LIN {X 0,Y 85.092,Z 662.145,A -85,B 0,C 180,E1 -19260,E2 -19260} C_VEL
LIN {X 0,Y 82.848,Z 665.659,A -85,B 0,C 180,E1 -19250.232,E2 -19250.232} C_VEL
LIN {X 0,Y 84.77,Z 669.976,A -85,B 0,C 180,E1 -19235.51,E2 -19235.51} C_VEL
LIN {X 0,Y 86.766,Z 671.167,A -85,B 0,C 180,E1 -19230.922,E2 -19230.922} C_VEL
LIN {X 0,Y 92.025,Z 672.605,A -85,B 0,C 180,E1 -19223.904,E2 -19223.904} C_VEL
LIN {X 0,Y 91.235,Z 673.792,A -85,B 0,C 180,E1 -19222.952,E2 -19222.952} C_VEL
LIN {X 0,Y 83.813,Z 680.743,A -85,B 0,C 180,E1 -19217.869,E2 -19217.869} C_VEL
LIN {X 0,Y 77.915,Z 685.734,A -85,B 0,C 180,E1 -19212.572,E2 -19212.572} C_VEL
LIN {X 0,Y 72.15,Z 690.144,A -85,B 0,C 180,E1 -19205.764,E2 -19205.764} C_VEL
LIN {X 0,Y 68.908,Z 692.468,A -85,B 0,C 180,E1 -19200.661,E2 -19200.661} C_VEL
LIN {X 0,Y 66.35,Z 694.368,A -85,B 0,C 180,E1 -19195.068,E2 -19195.068} C_VEL
LIN {X 0,Y 64.456,Z 695.815,A -85,B 0,C 180,E1 -19189.093,E2 -19189.093} C_VEL
LIN {X 0,Y 63.195,Z 696.835,A -85,B 0,C 180,E1 -19182.851,E2 -19182.851} C_VEL
LIN {X 0,Y 62.592,Z 697.466,A -85,B 0,C 180,E1 -19176.447,E2 -19176.447} C_VEL
LIN {X 0,Y 62.642,Z 697.705,A -85,B 0,C 180,E1 -19170,E2 -19170} C_VEL
LIN {X 0,Y 62.755,Z 697.489,A -85,B 0,C 180,E1 -19163.57,E2 -19163.57} C_VEL
LIN {X 0,Y 64.913,Z 695.872,A -85,B 0,C 180,E1 -19151.046,E2 -19151.046} C_VEL
LIN {X 0,Y 67.088,Z 694.459,A -85,B 0,C 180,E1 -19145.226,E2 -19145.226} C_VEL
LIN {X 0,Y 71.596,Z 691.514,A -85,B 0,C 180,E1 -19137.324,E2 -19137.324} C_VEL
LIN {X 0,Y 77.419,Z 687.523,A -85,B 0,C 180,E1 -19130.546,E2 -19130.546} C_VEL
LIN {X 0,Y 84.572,Z 682.371,A -85,B 0,C 180,E1 -19125.06,E2 -19125.06} C_VEL
LIN {X 0,Y 87.182,Z 680.379,A -85,B 0,C 180,E1 -19123.488,E2 -19123.488} C_VEL
LIN {X 0,Y 82.264,Z 678.447,A -85,B 0,C 180,E1 -19116.729,E2 -19116.729} C_VEL
LIN {X 0,Y 79.03,Z 677.694,A -85,B 0,C 180,E1 -19112.247,E2 -19112.247} C_VEL
LIN {X 0,Y 76.795,Z 676.602,A -85,B 0,C 180,E1 -19107.231,E2 -19107.231} C_VEL
LIN {X 0,Y 75.533,Z 675.043,A -85,B 0,C 180,E1 -19101.494,E2 -19101.494} C_VEL
LIN {X 0,Y 74.478,Z 672.702,A -85,B 0,C 180,E1 -19090.878,E2 -19090.878} C_VEL
LIN {X 0,Y 76.565,Z 669.743,A -85,B 0,C 180,E1 -19080,E2 -19080} C_VEL
LIN {X 0,Y 83.879,Z 665.425,A -85,B 0,C 180,E1 -19065.442,E2 -19065.442} C_VEL
LIN {X 0,Y 96.513,Z 659.738,A -85,B 0,C 180,E1 -19054.092,E2 -19054.092} C_VEL
LIN {X 0,Y 99.35,Z 658.243,A -85,B 0,C 180,E1 -19052.625,E2 -19052.625} C_VEL
LIN {X 0,Y 105.136,Z 655.722,A -85,B 0,C 180,E1 -19049.405,E2 -19049.405} C_VEL
LIN {X 0,Y 105.017,Z 656.515,A -85,B 0,C 180,E1 -19048.696,E2 -19048.696} C_VEL
LIN {X 0,Y 98.158,Z 664.839,A -85,B 0,C 180,E1 -19045.426,E2 -19045.426} C_VEL
LIN {X 0,Y 90.491,Z 672.846,A -85,B 0,C 180,E1 -19040.955,E2 -19040.955} C_VEL
LIN {X 0,Y 83.376,Z 679.286,A -85,B 0,C 180,E1 -19035.766,E2 -19035.766} C_VEL
LIN {X 0,Y 76.898,Z 684.398,A -85,B 0,C 180,E1 -19029.774,E2 -19029.774} C_VEL
LIN {X 0,Y 71.412,Z 688.419,A -85,B 0,C 180,E1 -19022.496,E2 -19022.496} C_VEL
LIN {X 0,Y 68.389,Z 690.108,A -85,B 0,C 180,E1 -19018.544,E2 -19018.544} C_VEL
LIN {X 0,Y 62.458,Z 692.322,A -85,B 0,C 180,E1 -19011.839,E2 -19011.839} C_VEL
LIN {X 0,Y 58.208,Z 693.565,A -85,B 0,C 180,E1 -19005.545,E2 -19005.545} C_VEL
LIN {X 0,Y 56.215,Z 694.173,A -85,B 0,C 180,E1 -18999.984,E2 -18999.984} C_VEL
LIN {X 0,Y 55.916,Z 694.293,A -85,B 0,C 180,E1 -18997.996,E2 -18997.996} C_VEL
LIN {X 0,Y 55.609,Z 694.556,A -85,B 0,C 180,E1 -18990,E2 -18990} C_VEL
LIN {X 0,Y 56.865,Z 693.723,A -85,B 0,C 180,E1 -18975.689,E2 -18975.689} C_VEL
LIN {X 0,Y 58.571,Z 692.733,A -85,B 0,C 180,E1 -18968.901,E2 -18968.901} C_VEL
LIN {X 0,Y 60.958,Z 691.321,A -85,B 0,C 180,E1 -18962.537,E2 -18962.537} C_VEL
LIN {X 0,Y 65.7,Z 688.393,A -85,B 0,C 180,E1 -18953.961,E2 -18953.961} C_VEL
LIN {X 0,Y 71.617,Z 684.415,A -85,B 0,C 180,E1 -18946.612,E2 -18946.612} C_VEL
LIN {X 0,Y 78.615,Z 679.262,A -85,B 0,C 180,E1 -18940.546,E2 -18940.546} C_VEL
LIN {X 0,Y 86.232,Z 672.778,A -85,B 0,C 180,E1 -18935.412,E2 -18935.412} C_VEL
LIN {X 0,Y 94.349,Z 664.71,A -85,B 0,C 180,E1 -18931.059,E2 -18931.059} C_VEL
LIN {X 0,Y 101.472,Z 656.423,A -85,B 0,C 180,E1 -18927.984,E2 -18927.984} C_VEL
LIN {X 0,Y 105.069,Z 651.685,A -85,B 0,C 180,E1 -18926.643,E2 -18926.643} C_VEL
LIN {X 0,Y 105.974,Z 649.829,A -85,B 0,C 180,E1 -18925.697,E2 -18925.697} C_VEL
LIN {X 0,Y 97.243,Z 655.594,A -85,B 0,C 180,E1 -18921.184,E2 -18921.184} C_VEL
LIN {X 0,Y 92.45,Z 658.477,A -85,B 0,C 180,E1 -18917.703,E2 -18917.703} C_VEL
LIN {X 0,Y 88.64,Z 660.634,A -85,B 0,C 180,E1 -18913.761,E2 -18913.761} C_VEL
LIN {X 0,Y 85.467,Z 662.497,A -85,B 0,C 180,E1 -18909.466,E2 -18909.466} C_VEL
LIN {X 0,Y 80.521,Z 666.215,A -85,B 0,C 180,E1 -18902.501,E2 -18902.501} C_VEL
LIN {X 0,Y 77.739,Z 669.133,A -85,B 0,C 180,E1 -18893.966,E2 -18893.966} C_VEL
LIN {X 0,Y 80.998,Z 675.167,A -85,B 0,C 180,E1 -18870.191,E2 -18870.191} C_VEL
LIN {X 0,Y 83.783,Z 675.989,A -85,B 0,C 180,E1 -18865.868,E2 -18865.868} C_VEL
LIN {X 0,Y 82.502,Z 677.724,A -85,B 0,C 180,E1 -18864.025,E2 -18864.025} C_VEL
LIN {X 0,Y 75.151,Z 683.798,A -85,B 0,C 180,E1 -18858.431,E2 -18858.431} C_VEL
LIN {X 0,Y 68.463,Z 688.599,A -85,B 0,C 180,E1 -18851.856,E2 -18851.856} C_VEL
LIN {X 0,Y 62.89,Z 692.278,A -85,B 0,C 180,E1 -18843.97,E2 -18843.97} C_VEL
LIN {X 0,Y 59.952,Z 694.177,A -85,B 0,C 180,E1 -18837.964,E2 -18837.964} C_VEL
LIN {X 0,Y 57.765,Z 695.625,A -85,B 0,C 180,E1 -18831.408,E2 -18831.408} C_VEL
LIN {X 0,Y 56.28,Z 696.646,A -85,B 0,C 180,E1 -18824.463,E2 -18824.463} C_VEL
LIN {X 0,Y 55.542,Z 697.277,A -85,B 0,C 180,E1 -18817.269,E2 -18817.269} C_VEL
LIN {X 0,Y 55.532,Z 697.516,A -85,B 0,C 180,E1 -18810,E2 -18810} C_VEL
LIN {X 0,Y 55.692,Z 697.3,A -85,B 0,C 180,E1 -18802.75,E2 -18802.75} C_VEL
LIN {X 0,Y 58.239,Z 695.683,A -85,B 0,C 180,E1 -18788.775,E2 -18788.775} C_VEL
LIN {X 0,Y 60.713,Z 694.271,A -85,B 0,C 180,E1 -18782.417,E2 -18782.417} C_VEL
LIN {X 0,Y 65.745,Z 691.327,A -85,B 0,C 180,E1 -18773.989,E2 -18773.989} C_VEL
LIN {X 0,Y 72.078,Z 687.336,A -85,B 0,C 180,E1 -18766.958,E2 -18766.958} C_VEL
LIN {X 0,Y 78.39,Z 683.096,A -85,B 0,C 180,E1 -18762.238,E2 -18762.238} C_VEL
LIN {X 0,Y 78.058,Z 682.451,A -85,B 0,C 180,E1 -18760.697,E2 -18760.697} C_VEL
LIN {X 0,Y 71.292,Z 680.424,A -85,B 0,C 180,E1 -18749.531,E2 -18749.531} C_VEL
LIN {X 0,Y 72.504,Z 672.841,A -85,B 0,C 180,E1 -18714.437,E2 -18714.437} C_VEL
LIN {X 0,Y 78.276,Z 670.097,A -85,B 0,C 180,E1 -18704.374,E2 -18704.374} C_VEL
LIN {X 0,Y 94.026,Z 663.899,A -85,B 0,C 180,E1 -18690.988,E2 -18690.988} C_VEL
LIN {X 0,Y 95.328,Z 663.283,A -85,B 0,C 180,E1 -18690.369,E2 -18690.369} C_VEL
LIN {X 0,Y 94.903,Z 664.393,A -85,B 0,C 180,E1 -18689.273,E2 -18689.273} C_VEL
LIN {X 0,Y 87.657,Z 671.706,A -85,B 0,C 180,E1 -18685.458,E2 -18685.458} C_VEL
LIN {X 0,Y 81.075,Z 677.49,A -85,B 0,C 180,E1 -18681.276,E2 -18681.276} C_VEL
LIN {X 0,Y 73.843,Z 683,A -85,B 0,C 180,E1 -18675.547,E2 -18675.547} C_VEL
LIN {X 0,Y 67.513,Z 687.308,A -85,B 0,C 180,E1 -18668.652,E2 -18668.652} C_VEL
LIN {X 0,Y 63.94,Z 689.573,A -85,B 0,C 180,E1 -18663.338,E2 -18663.338} C_VEL
LIN {X 0,Y 60.953,Z 691.413,A -85,B 0,C 180,E1 -18657.465,E2 -18657.465} C_VEL
LIN {X 0,Y 58.569,Z 692.792,A -85,B 0,C 180,E1 -18651.099,E2 -18651.099} C_VEL
LIN {X 0,Y 55.916,Z 694.293,A -85,B 0,C 180,E1 -18637.996,E2 -18637.996} C_VEL
LIN {X 0,Y 55.317,Z 694.556,A -85,B 0,C 180,E1 -18633.998,E2 -18633.998} C_VEL
LIN {X 0,Y 53.901,Z 694.702,A -85,B 0,C 180,E1 -18627.956,E2 -18627.956} C_VEL
LIN {X 0,Y 51.663,Z 694.275,A -85,B 0,C 180,E1 -18617.386,E2 -18617.386} C_VEL
LIN {X 0,Y 51.576,Z 693.301,A -85,B 0,C 180,E1 -18608.562,E2 -18608.562} C_VEL
LIN {X 0,Y 52.568,Z 692.593,A -85,B 0,C 180,E1 -18604.386,E2 -18604.386} C_VEL
LIN {X 0,Y 58.152,Z 689.651,A -85,B 0,C 180,E1 -18592.823,E2 -18592.823} C_VEL
LIN {X 0,Y 64.344,Z 686.033,A -85,B 0,C 180,E1 -18584.768,E2 -18584.768} C_VEL
LIN {X 0,Y 71.589,Z 681.293,A -85,B 0,C 180,E1 -18578.245,E2 -18578.245} C_VEL
LIN {X 0,Y 79.553,Z 675.292,A -85,B 0,C 180,E1 -18572.937,E2 -18572.937} C_VEL
LIN {X 0,Y 87.984,Z 667.809,A -85,B 0,C 180,E1 -18568.518,E2 -18568.518} C_VEL
LIN {X 0,Y 94.958,Z 660.558,A -85,B 0,C 180,E1 -18565.594,E2 -18565.594} C_VEL
LIN {X 0,Y 95.736,Z 659.289,A -85,B 0,C 180,E1 -18564.747,E2 -18564.747} C_VEL
LIN {X 0,Y 90.805,Z 661.951,A -85,B 0,C 180,E1 -18561.757,E2 -18561.757} C_VEL
LIN {X 0,Y 87.102,Z 663.828,A -85,B 0,C 180,E1 -18558.83,E2 -18558.83} C_VEL
LIN {X 0,Y 80.808,Z 666.963,A -85,B 0,C 180,E1 -18551.657,E2 -18551.657} C_VEL
LIN {X 0,Y 75.932,Z 670.038,A -85,B 0,C 180,E1 -18545.311,E2 -18545.311} C_VEL
LIN {X 0,Y 73.444,Z 671.868,A -85,B 0,C 180,E1 -18540,E2 -18540} C_VEL
LIN {X 0,Y 72.428,Z 677.195,A -85,B 0,C 180,E1 -18517.162,E2 -18517.162} C_VEL
LIN {X 0,Y 74.052,Z 678.364,A -85,B 0,C 180,E1 -18511.672,E2 -18511.672} C_VEL
LIN {X 0,Y 75.813,Z 679.737,A -85,B 0,C 180,E1 -18506.545,E2 -18506.545} C_VEL
LIN {X 0,Y 68.118,Z 685.355,A -85,B 0,C 180,E1 -18500.697,E2 -18500.697} C_VEL
LIN {X 0,Y 61.161,Z 689.764,A -85,B 0,C 180,E1 -18493.588,E2 -18493.588} C_VEL
LIN {X 0,Y 57.129,Z 692.088,A -85,B 0,C 180,E1 -18487.959,E2 -18487.959} C_VEL
LIN {X 0,Y 53.746,Z 693.986,A -85,B 0,C 180,E1 -18481.537,E2 -18481.537} C_VEL
LIN {X 0,Y 51.176,Z 695.434,A -85,B 0,C 180,E1 -18474.33,E2 -18474.33} C_VEL
LIN {X 0,Y 49.403,Z 696.455,A -85,B 0,C 180,E1 -18466.53,E2 -18466.53} C_VEL
LIN {X 0,Y 48.496,Z 697.087,A -85,B 0,C 180,E1 -18458.333,E2 -18458.333} C_VEL
LIN {X 0,Y 48.443,Z 697.327,A -85,B 0,C 180,E1 -18450,E2 -18450} C_VEL
LIN {X 0,Y 48.649,Z 697.111,A -85,B 0,C 180,E1 -18441.694,E2 -18441.694} C_VEL
LIN {X 0,Y 51.688,Z 695.495,A -85,B 0,C 180,E1 -18425.926,E2 -18425.926} C_VEL
LIN {X 0,Y 54.508,Z 694.083,A -85,B 0,C 180,E1 -18418.953,E2 -18418.953} C_VEL
LIN {X 0,Y 60.142,Z 691.139,A -85,B 0,C 180,E1 -18410.006,E2 -18410.006} C_VEL
LIN {X 0,Y 68.937,Z 685.995,A -85,B 0,C 180,E1 -18401.363,E2 -18401.363} C_VEL
LIN {X 0,Y 69.573,Z 684.914,A -85,B 0,C 180,E1 -18399.083,E2 -18399.083} C_VEL
LIN {X 0,Y 64.877,Z 683.489,A -85,B 0,C 180,E1 -18389.931,E2 -18389.931} C_VEL
LIN {X 0,Y 66.397,Z 676.925,A -85,B 0,C 180,E1 -18353.924,E2 -18353.924} C_VEL
LIN {X 0,Y 74.494,Z 673.684,A -85,B 0,C 180,E1 -18340.636,E2 -18340.636} C_VEL
LIN {X 0,Y 86.317,Z 669.604,A -85,B 0,C 180,E1 -18330.756,E2 -18330.756} C_VEL
LIN {X 0,Y 78.2,Z 676.613,A -85,B 0,C 180,E1 -18326.234,E2 -18326.234} C_VEL
LIN {X 0,Y 71.57,Z 681.48,A -85,B 0,C 180,E1 -18321.774,E2 -18321.774} C_VEL
LIN {X 0,Y 64.309,Z 686.182,A -85,B 0,C 180,E1 -18315.264,E2 -18315.264} C_VEL
LIN {X 0,Y 58.139,Z 689.761,A -85,B 0,C 180,E1 -18307.187,E2 -18307.187} C_VEL
LIN {X 0,Y 54.735,Z 691.601,A -85,B 0,C 180,E1 -18300.904,E2 -18300.904} C_VEL
LIN {X 0,Y 51.998,Z 692.98,A -85,B 0,C 180,E1 -18293.921,E2 -18293.921} C_VEL
LIN {X 0,Y 48.876,Z 694.508,A -85,B 0,C 180,E1 -18278.791,E2 -18278.791} C_VEL
LIN {X 0,Y 48.509,Z 694.745,A -85,B 0,C 180,E1 -18270,E2 -18270} C_VEL
LIN {X 0,Y 48.83,Z 694.52,A -85,B 0,C 180,E1 -18261.725,E2 -18261.725} C_VEL
LIN {X 0,Y 50.014,Z 693.912,A -85,B 0,C 180,E1 -18253.677,E2 -18253.677} C_VEL
LIN {X 0,Y 52.568,Z 692.593,A -85,B 0,C 180,E1 -18244.386,E2 -18244.386} C_VEL
LIN {X 0,Y 54.273,Z 691.458,A -85,B 0,C 180,E1 -18238.45,E2 -18238.45} C_VEL
LIN {X 0,Y 56.572,Z 689.104,A -85,B 0,C 180,E1 -18228.741,E2 -18228.741} C_VEL
LIN {X 0,Y 60.191,Z 686.092,A -85,B 0,C 180,E1 -18220.151,E2 -18220.151} C_VEL
LIN {X 0,Y 63.687,Z 683.821,A -85,B 0,C 180,E1 -18216.265,E2 -18216.265} C_VEL
LIN {X 0,Y 73.054,Z 677.657,A -85,B 0,C 180,E1 -18210.023,E2 -18210.023} C_VEL
LIN {X 0,Y 81.588,Z 670.891,A -85,B 0,C 180,E1 -18205.734,E2 -18205.734} C_VEL
LIN {X 0,Y 84.818,Z 667.997,A -85,B 0,C 180,E1 -18204.293,E2 -18204.293} C_VEL
LIN {X 0,Y 85.518,Z 667.032,A -85,B 0,C 180,E1 -18203.369,E2 -18203.369} C_VEL
LIN {X 0,Y 75.4,Z 671.494,A -85,B 0,C 180,E1 -18193.476,E2 -18193.476} C_VEL
LIN {X 0,Y 69.774,Z 674.51,A -85,B 0,C 180,E1 -18185.781,E2 -18185.781} C_VEL
LIN {X 0,Y 65.852,Z 677.434,A -85,B 0,C 180,E1 -18173.874,E2 -18173.874} C_VEL
LIN {X 0,Y 68.399,Z 682.147,A -85,B 0,C 180,E1 -18149.086,E2 -18149.086} C_VEL
LIN {X 0,Y 61.18,Z 686.77,A -85,B 0,C 180,E1 -18143.526,E2 -18143.526} C_VEL
LIN {X 0,Y 53.884,Z 690.812,A -85,B 0,C 180,E1 -18135.837,E2 -18135.837} C_VEL
LIN {X 0,Y 47.806,Z 693.796,A -85,B 0,C 180,E1 -18126.018,E2 -18126.018} C_VEL
LIN {X 0,Y 44.768,Z 695.244,A -85,B 0,C 180,E1 -18118.097,E2 -18118.097} C_VEL
LIN {X 0,Y 42.618,Z 696.265,A -85,B 0,C 180,E1 -18109.257,E2 -18109.257} C_VEL
LIN {X 0,Y 41.465,Z 696.897,A -85,B 0,C 180,E1 -18099.758,E2 -18099.758} C_VEL
LIN {X 0,Y 41.338,Z 697.138,A -85,B 0,C 180,E1 -18090,E2 -18090} C_VEL
LIN {X 0,Y 41.643,Z 696.922,A -85,B 0,C 180,E1 -18080.284,E2 -18080.284} C_VEL
LIN {X 0,Y 45.307,Z 695.307,A -85,B 0,C 180,E1 -18062.267,E2 -18062.267} C_VEL
LIN {X 0,Y 48.554,Z 693.894,A -85,B 0,C 180,E1 -18054.621,E2 -18054.621} C_VEL
LIN {X 0,Y 54.893,Z 690.951,A -85,B 0,C 180,E1 -18045.237,E2 -18045.237} C_VEL
LIN {X 0,Y 59.784,Z 688.424,A -85,B 0,C 180,E1 -18040.288,E2 -18040.288} C_VEL
LIN {X 0,Y 61.088,Z 687.141,A -85,B 0,C 180,E1 -18037.159,E2 -18037.159} C_VEL
LIN {X 0,Y 57.929,Z 686.032,A -85,B 0,C 180,E1 -18029.031,E2 -18029.031} C_VEL
LIN {X 0,Y 62.933,Z 679.529,A -85,B 0,C 180,E1 -17987.094,E2 -17987.094} C_VEL
LIN {X 0,Y 70.775,Z 677.049,A -85,B 0,C 180,E1 -17976.596,E2 -17976.596} C_VEL
LIN {X 0,Y 75.71,Z 675.543,A -85,B 0,C 180,E1 -17972.345,E2 -17972.345} C_VEL
LIN {X 0,Y 75.018,Z 676.379,A -85,B 0,C 180,E1 -17971.111,E2 -17971.111} C_VEL
LIN {X 0,Y 67.412,Z 681.666,A -85,B 0,C 180,E1 -17966.516,E2 -17966.516} C_VEL
LIN {X 0,Y 59.527,Z 686.369,A -85,B 0,C 180,E1 -17960.122,E2 -17960.122} C_VEL
LIN {X 0,Y 52.661,Z 689.948,A -85,B 0,C 180,E1 -17951.858,E2 -17951.858} C_VEL
LIN {X 0,Y 48.772,Z 691.79,A -85,B 0,C 180,E1 -17945.198,E2 -17945.198} C_VEL
LIN {X 0,Y 45.597,Z 693.169,A -85,B 0,C 180,E1 -17937.542,E2 -17937.542} C_VEL
LIN {X 0,Y 41.827,Z 694.733,A -85,B 0,C 180,E1 -17919.673,E2 -17919.673} C_VEL
LIN {X 0,Y 41.428,Z 694.933,A -85,B 0,C 180,E1 -17910,E2 -17910} C_VEL
LIN {X 0,Y 41.827,Z 694.709,A -85,B 0,C 180,E1 -17900.327,E2 -17900.327} C_VEL
LIN {X 0,Y 45.599,Z 693.112,A -85,B 0,C 180,E1 -17882.459,E2 -17882.459} C_VEL
LIN {X 0,Y 48.777,Z 691.701,A -85,B 0,C 180,E1 -17874.807,E2 -17874.807} C_VEL
LIN {X 0,Y 54.859,Z 688.772,A -85,B 0,C 180,E1 -17865.202,E2 -17865.202} C_VEL
LIN {X 0,Y 63.687,Z 683.821,A -85,B 0,C 180,E1 -17856.265,E2 -17856.265} C_VEL
LIN {X 0,Y 65.986,Z 682.207,A -85,B 0,C 180,E1 -17853.77,E2 -17853.77} C_VEL
LIN {X 0,Y 68.675,Z 679.563,A -85,B 0,C 180,E1 -17848.988,E2 -17848.988} C_VEL
LIN {X 0,Y 71.665,Z 676.674,A -85,B 0,C 180,E1 -17844.636,E2 -17844.636} C_VEL
LIN {X 0,Y 74.25,Z 674.606,A -85,B 0,C 180,E1 -17842.878,E2 -17842.878} C_VEL
LIN {X 0,Y 75.901,Z 673.342,A -85,B 0,C 180,E1 -17842.188,E2 -17842.188} C_VEL
LIN {X 0,Y 75.893,Z 673.209,A -85,B 0,C 180,E1 -17841.742,E2 -17841.742} C_VEL
LIN {X 0,Y 71.385,Z 674.973,A -85,B 0,C 180,E1 -17837.179,E2 -17837.179} C_VEL
LIN {X 0,Y 66.86,Z 676.944,A -85,B 0,C 180,E1 -17832.136,E2 -17832.136} C_VEL
LIN {X 0,Y 60.935,Z 679.942,A -85,B 0,C 180,E1 -17820,E2 -17820} C_VEL
LIN {X 0,Y 60.784,Z 684.404,A -85,B 0,C 180,E1 -17792.452,E2 -17792.452} C_VEL
LIN {X 0,Y 59.15,Z 685.508,A -85,B 0,C 180,E1 -17790.623,E2 -17790.623} C_VEL
LIN {X 0,Y 49.184,Z 690.621,A -85,B 0,C 180,E1 -17781.805,E2 -17781.805} C_VEL
LIN {X 0,Y 42.242,Z 693.605,A -85,B 0,C 180,E1 -17771.721,E2 -17771.721} C_VEL
LIN {X 0,Y 38.624,Z 695.054,A -85,B 0,C 180,E1 -17763.084,E2 -17763.084} C_VEL
LIN {X 0,Y 35.976,Z 696.075,A -85,B 0,C 180,E1 -17752.999,E2 -17752.999} C_VEL
LIN {X 0,Y 34.483,Z 696.708,A -85,B 0,C 180,E1 -17741.76,E2 -17741.76} C_VEL
LIN {X 0,Y 34.25,Z 696.949,A -85,B 0,C 180,E1 -17730,E2 -17730} C_VEL
LIN {X 0,Y 34.661,Z 696.733,A -85,B 0,C 180,E1 -17718.301,E2 -17718.301} C_VEL
LIN {X 0,Y 39.15,Z 695.118,A -85,B 0,C 180,E1 -17697.415,E2 -17697.415} C_VEL
LIN {X 0,Y 42.96,Z 693.706,A -85,B 0,C 180,E1 -17689.128,E2 -17689.128} C_VEL
LIN {X 0,Y 50.104,Z 690.764,A -85,B 0,C 180,E1 -17679.513,E2 -17679.513} C_VEL
LIN {X 0,Y 52.741,Z 689.535,A -85,B 0,C 180,E1 -17676.914,E2 -17676.914} C_VEL
LIN {X 0,Y 52.116,Z 688.831,A -85,B 0,C 180,E1 -17672.644,E2 -17672.644} C_VEL
LIN {X 0,Y 59.574,Z 682.124,A -85,B 0,C 180,E1 -17620.694,E2 -17620.694} C_VEL
LIN {X 0,Y 65.544,Z 680.589,A -85,B 0,C 180,E1 -17613.688,E2 -17613.688} C_VEL
LIN {X 0,Y 64.735,Z 681.272,A -85,B 0,C 180,E1 -17612.397,E2 -17612.397} C_VEL
LIN {X 0,Y 55.233,Z 686.557,A -85,B 0,C 180,E1 -17605.8,E2 -17605.8} C_VEL
LIN {X 0,Y 47.598,Z 690.136,A -85,B 0,C 180,E1 -17597.584,E2 -17597.584} C_VEL
LIN {X 0,Y 43.165,Z 691.978,A -85,B 0,C 180,E1 -17590.638,E2 -17590.638} C_VEL
LIN {X 0,Y 39.445,Z 693.357,A -85,B 0,C 180,E1 -17582.312,E2 -17582.312} C_VEL
LIN {X 0,Y 34.844,Z 694.922,A -85,B 0,C 180,E1 -17561.636,E2 -17561.636} C_VEL
LIN {X 0,Y 34.33,Z 695.122,A -85,B 0,C 180,E1 -17550,E2 -17550} C_VEL
LIN {X 0,Y 34.844,Z 694.898,A -85,B 0,C 180,E1 -17538.364,E2 -17538.364} C_VEL
LIN {X 0,Y 39.447,Z 693.301,A -85,B 0,C 180,E1 -17517.69,E2 -17517.69} C_VEL
LIN {X 0,Y 43.17,Z 691.89,A -85,B 0,C 180,E1 -17509.368,E2 -17509.368} C_VEL
LIN {X 0,Y 50.055,Z 688.962,A -85,B 0,C 180,E1 -17499.446,E2 -17499.446} C_VEL
LIN {X 0,Y 59.427,Z 684.198,A -85,B 0,C 180,E1 -17491.011,E2 -17491.011} C_VEL
LIN {X 0,Y 69.769,Z 677.845,A -85,B 0,C 180,E1 -17484.961,E2 -17484.961} C_VEL
LIN {X 0,Y 74.25,Z 674.606,A -85,B 0,C 180,E1 -17482.878,E2 -17482.878} C_VEL
LIN {X 0,Y 74.636,Z 674.135,A -85,B 0,C 180,E1 -17482.046,E2 -17482.046} C_VEL
LIN {X 0,Y 73.873,Z 674.135,A -85,B 0,C 180,E1 -17480.257,E2 -17480.257} C_VEL
LIN {X 0,Y 71.107,Z 675.24,A -85,B 0,C 180,E1 -17477.583,E2 -17477.583} C_VEL
LIN {X 0,Y 68.611,Z 676.406,A -85,B 0,C 180,E1 -17475.766,E2 -17475.766} C_VEL
LIN {X 0,Y 58.828,Z 681.238,A -85,B 0,C 180,E1 -17468.369,E2 -17468.369} C_VEL
LIN {X 0,Y 55.87,Z 682.623,A -85,B 0,C 180,E1 -17464.137,E2 -17464.137} C_VEL
LIN {X 0,Y 54.855,Z 683.138,A -85,B 0,C 180,E1 -17461.638,E2 -17461.638} C_VEL
LIN {X 0,Y 53.298,Z 686.474,A -85,B 0,C 180,E1 -17436.698,E2 -17436.698} C_VEL
LIN {X 0,Y 50.804,Z 687.889,A -85,B 0,C 180,E1 -17433.736,E2 -17433.736} C_VEL
LIN {X 0,Y 42.36,Z 691.518,A -85,B 0,C 180,E1 -17426.054,E2 -17426.054} C_VEL
LIN {X 0,Y 37.218,Z 693.415,A -85,B 0,C 180,E1 -17419.055,E2 -17419.055} C_VEL
LIN {X 0,Y 32.887,Z 694.864,A -85,B 0,C 180,E1 -17409.874,E2 -17409.874} C_VEL
LIN {X 0,Y 27.55,Z 696.518,A -85,B 0,C 180,E1 -17384.779,E2 -17384.779} C_VEL
LIN {X 0,Y 27.136,Z 696.76,A -85,B 0,C 180,E1 -17370,E2 -17370} C_VEL
LIN {X 0,Y 27.735,Z 696.544,A -85,B 0,C 180,E1 -17355.321,E2 -17355.321} C_VEL
LIN {X 0,Y 33.383,Z 694.929,A -85,B 0,C 180,E1 -17330.833,E2 -17330.833} C_VEL
LIN {X 0,Y 37.879,Z 693.518,A -85,B 0,C 180,E1 -17322.085,E2 -17322.085} C_VEL
LIN {X 0,Y 44.349,Z 691.173,A -85,B 0,C 180,E1 -17314.133,E2 -17314.133} C_VEL
LIN {X 0,Y 44.667,Z 690.651,A -85,B 0,C 180,E1 -17311.022,E2 -17311.022} C_VEL
LIN {X 0,Y 54.168,Z 685.081,A -85,B 0,C 180,E1 -17257.093,E2 -17257.093} C_VEL
LIN {X 0,Y 54.582,Z 685.33,A -85,B 0,C 180,E1 -17254.332,E2 -17254.332} C_VEL
LIN {X 0,Y 45.838,Z 689.272,A -85,B 0,C 180,E1 -17247.488,E2 -17247.488} C_VEL
LIN {X 0,Y 38.063,Z 692.166,A -85,B 0,C 180,E1 -17237.61,E2 -17237.61} C_VEL
LIN {X 0,Y 33.645,Z 693.546,A -85,B 0,C 180,E1 -17228.804,E2 -17228.804} C_VEL
LIN {X 0,Y 30.178,Z 694.52,A -85,B 0,C 180,E1 -17217.761,E2 -17217.761} C_VEL
LIN {X 0,Y 27.931,Z 695.111,A -85,B 0,C 180,E1 -17204.573,E2 -17204.573} C_VEL
LIN {X 0,Y 27.248,Z 695.311,A -85,B 0,C 180,E1 -17190,E2 -17190} C_VEL
LIN {X 0,Y 30.178,Z 694.48,A -85,B 0,C 180,E1 -17162.24,E2 -17162.24} C_VEL
LIN {X 0,Y 33.647,Z 693.491,A -85,B 0,C 180,E1 -17151.199,E2 -17151.199} C_VEL
LIN {X 0,Y 38.069,Z 692.079,A -85,B 0,C 180,E1 -17142.4,E2 -17142.4} C_VEL
LIN {X 0,Y 45.864,Z 689.152,A -85,B 0,C 180,E1 -17132.563,E2 -17132.563} C_VEL
LIN {X 0,Y 54.596,Z 685.171,A -85,B 0,C 180,E1 -17125.698,E2 -17125.698} C_VEL
LIN {X 0,Y 63.106,Z 680.521,A -85,B 0,C 180,E1 -17121.193,E2 -17121.193} C_VEL
LIN {X 0,Y 64.967,Z 679.09,A -85,B 0,C 180,E1 -17118.938,E2 -17118.938} C_VEL
LIN {X 0,Y 60.419,Z 680.796,A -85,B 0,C 180,E1 -17113.453,E2 -17113.453} C_VEL
LIN {X 0,Y 54.855,Z 683.138,A -85,B 0,C 180,E1 -17101.638,E2 -17101.638} C_VEL
LIN {X 0,Y 52.902,Z 684.251,A -85,B 0,C 180,E1 -17096.504,E2 -17096.504} C_VEL
LIN {X 0,Y 50.501,Z 685.667,A -85,B 0,C 180,E1 -17091.444,E2 -17091.444} C_VEL
LIN {X 0,Y 45.399,Z 688.751,A -85,B 0,C 180,E1 -17080.577,E2 -17080.577} C_VEL
LIN {X 0,Y 45.001,Z 689.002,A -85,B 0,C 180,E1 -17079.561,E2 -17079.561} C_VEL
LIN {X 0,Y 38.833,Z 691.328,A -85,B 0,C 180,E1 -17074.811,E2 -17074.811} C_VEL
LIN {X 0,Y 32.984,Z 693.224,A -85,B 0,C 180,E1 -17068.462,E2 -17068.462} C_VEL
LIN {X 0,Y 27.789,Z 694.673,A -85,B 0,C 180,E1 -17059.352,E2 -17059.352} C_VEL
LIN {X 0,Y 20.755,Z 696.329,A -85,B 0,C 180,E1 -17029.793,E2 -17029.793} C_VEL
LIN {X 0,Y 20.026,Z 696.57,A -85,B 0,C 180,E1 -17010,E2 -17010} C_VEL
LIN {X 0,Y 20.947,Z 696.355,A -85,B 0,C 180,E1 -16990.396,E2 -16990.396} C_VEL
LIN {X 0,Y 28.238,Z 694.741,A -85,B 0,C 180,E1 -16961.699,E2 -16961.699} C_VEL
LIN {X 0,Y 35.794,Z 692.634,A -85,B 0,C 180,E1 -16950.422,E2 -16950.422} C_VEL
LIN {X 0,Y 36.439,Z 691.812,A -85,B 0,C 180,E1 -16942.689,E2 -16942.689} C_VEL
LIN {X 0,Y 44.586,Z 688.45,A -85,B 0,C 180,E1 -16899.221,E2 -16899.221} C_VEL
LIN {X 0,Y 42.03,Z 689.61,A -85,B 0,C 180,E1 -16895.277,E2 -16895.277} C_VEL
LIN {X 0,Y 33.683,Z 692.354,A -85,B 0,C 180,E1 -16886.575,E2 -16886.575} C_VEL
LIN {X 0,Y 28.458,Z 693.735,A -85,B 0,C 180,E1 -16877.807,E2 -16877.807} C_VEL
LIN {X 0,Y 24.118,Z 694.709,A -85,B 0,C 180,E1 -16865.648,E2 -16865.648} C_VEL
LIN {X 0,Y 21.152,Z 695.3,A -85,B 0,C 180,E1 -16849.406,E2 -16849.406} C_VEL
LIN {X 0,Y 20.159,Z 695.5,A -85,B 0,C 180,E1 -16830,E2 -16830} C_VEL
LIN {X 0,Y 21.152,Z 695.276,A -85,B 0,C 180,E1 -16810.594,E2 -16810.594} C_VEL
LIN {X 0,Y 24.118,Z 694.67,A -85,B 0,C 180,E1 -16794.353,E2 -16794.353} C_VEL
LIN {X 0,Y 28.46,Z 693.681,A -85,B 0,C 180,E1 -16782.197,E2 -16782.197} C_VEL
LIN {X 0,Y 33.689,Z 692.269,A -85,B 0,C 180,E1 -16773.441,E2 -16773.441} C_VEL
LIN {X 0,Y 42.462,Z 689.342,A -85,B 0,C 180,E1 -16764.451,E2 -16764.451} C_VEL
LIN {X 0,Y 53.619,Z 684.525,A -85,B 0,C 180,E1 -16757.825,E2 -16757.825} C_VEL
LIN {X 0,Y 54.533,Z 683.959,A -85,B 0,C 180,E1 -16756.222,E2 -16756.222} C_VEL
LIN {X 0,Y 47.628,Z 686.461,A -85,B 0,C 180,E1 -16740,E2 -16740} C_VEL
LIN {X 0,Y 46.1,Z 688.327,A -85,B 0,C 180,E1 -16722.248,E2 -16722.248} C_VEL
LIN {X 0,Y 45.399,Z 688.751,A -85,B 0,C 180,E1 -16720.577,E2 -16720.577} C_VEL
LIN {X 0,Y 43.473,Z 689.734,A -85,B 0,C 180,E1 -16717.475,E2 -16717.475} C_VEL
LIN {X 0,Y 40.065,Z 691.035,A -85,B 0,C 180,E1 -16714.549,E2 -16714.549} C_VEL
LIN {X 0,Y 36.482,Z 692.133,A -85,B 0,C 180,E1 -16712.645,E2 -16712.645} C_VEL
LIN {X 0,Y 28.523,Z 693.9,A -85,B 0,C 180,E1 -16709.843,E2 -16709.843} C_VEL
LIN {X 0,Y 22.325,Z 694.945,A -85,B 0,C 180,E1 -16706.165,E2 -16706.165} C_VEL
LIN {X 0,Y 17.799,Z 695.595,A -85,B 0,C 180,E1 -16698.288,E2 -16698.288} C_VEL
LIN {X 0,Y 17.068,Z 695.67,A -85,B 0,C 180,E1 -16695.762,E2 -16695.762} C_VEL
LIN {X 0,Y 12.931,Z 696.381,A -85,B 0,C 180,E1 -16650,E2 -16650} C_VEL
LIN {X 0,Y 14.467,Z 696.167,A -85,B 0,C 180,E1 -16620.935,E2 -16620.935} C_VEL
LIN {X 0,Y 24.11,Z 694.552,A -85,B 0,C 180,E1 -16589.015,E2 -16589.015} C_VEL
LIN {X 0,Y 28.676,Z 693.521,A -85,B 0,C 180,E1 -16583.212,E2 -16583.212} C_VEL
LIN {X 0,Y 29.226,Z 692.968,A -85,B 0,C 180,E1 -16573.914,E2 -16573.914} C_VEL
LIN {X 0,Y 34.142,Z 691.405,A -85,B 0,C 180,E1 -16544.315,E2 -16544.315} C_VEL
LIN {X 0,Y 33.57,Z 691.655,A -85,B 0,C 180,E1 -16540.685,E2 -16540.685} C_VEL
LIN {X 0,Y 24.267,Z 693.923,A -85,B 0,C 180,E1 -16530.322,E2 -16530.322} C_VEL
LIN {X 0,Y 18.813,Z 694.897,A -85,B 0,C 180,E1 -16518.345,E2 -16518.345} C_VEL
LIN {X 0,Y 14.65,Z 695.488,A -85,B 0,C 180,E1 -16498.667,E2 -16498.667} C_VEL
LIN {X 0,Y 13.06,Z 695.689,A -85,B 0,C 180,E1 -16470,E2 -16470} C_VEL
LIN {X 0,Y 14.65,Z 695.465,A -85,B 0,C 180,E1 -16441.333,E2 -16441.333} C_VEL
LIN {X 0,Y 18.813,Z 694.859,A -85,B 0,C 180,E1 -16421.656,E2 -16421.656} C_VEL
LIN {X 0,Y 24.269,Z 693.87,A -85,B 0,C 180,E1 -16409.684,E2 -16409.684} C_VEL
LIN {X 0,Y 30.353,Z 692.459,A -85,B 0,C 180,E1 -16402.154,E2 -16402.154} C_VEL
LIN {X 0,Y 40.041,Z 689.532,A -85,B 0,C 180,E1 -16395.122,E2 -16395.122} C_VEL
LIN {X 0,Y 43.354,Z 688.315,A -85,B 0,C 180,E1 -16393.433,E2 -16393.433} C_VEL
LIN {X 0,Y 43.315,Z 688.196,A -85,B 0,C 180,E1 -16389.338,E2 -16389.338} C_VEL
LIN {X 0,Y 39.425,Z 689.949,A -85,B 0,C 180,E1 -16369.732,E2 -16369.732} C_VEL
LIN {X 0,Y 38.098,Z 690.585,A -85,B 0,C 180,E1 -16366.007,E2 -16366.007} C_VEL
LIN {X 0,Y 29.879,Z 693.034,A -85,B 0,C 180,E1 -16360.197,E2 -16360.197} C_VEL
LIN {X 0,Y 23.759,Z 694.483,A -85,B 0,C 180,E1 -16352.552,E2 -16352.552} C_VEL
LIN {X 0,Y 17.068,Z 695.67,A -85,B 0,C 180,E1 -16335.762,E2 -16335.762} C_VEL
LIN {X 0,Y 13.273,Z 696.165,A -85,B 0,C 180,E1 -16318.569,E2 -16318.569} C_VEL
LIN {X 0,Y 10.256,Z 696.3,A -85,B 0,C 180,E1 -16293.156,E2 -16293.156} C_VEL
LIN {X 0,Y 12.525,Z 695.741,A -85,B 0,C 180,E1 -16230.233,E2 -16230.233} C_VEL
LIN {X 0,Y 18.282,Z 694.917,A -85,B 0,C 180,E1 -16215.335,E2 -16215.335} C_VEL
LIN {X 0,Y 19.219,Z 694.714,A -85,B 0,C 180,E1 -16214.312,E2 -16214.312} C_VEL
LIN {X 0,Y 21.578,Z 694.364,A -85,B 0,C 180,E1 -16212.284,E2 -16212.284} C_VEL
LIN {X 0,Y 23.104,Z 693.886,A -85,B 0,C 180,E1 -16199.999,E2 -16199.999} C_VEL
LIN {X 0,Y 24.372,Z 693.586,A -85,B 0,C 180,E1 -16191.446,E2 -16191.446} C_VEL
LIN {X 0,Y 22.931,Z 693.894,A -85,B 0,C 180,E1 -16187.946,E2 -16187.946} C_VEL
LIN {X 0,Y 15.055,Z 695.086,A -85,B 0,C 180,E1 -16179.007,E2 -16179.007} C_VEL
LIN {X 0,Y 9.081,Z 695.677,A -85,B 0,C 180,E1 -16160.708,E2 -16160.708} C_VEL
LIN {X 0,Y 5.966,Z 695.878,A -85,B 0,C 180,E1 -16110,E2 -16110} C_VEL
LIN {X 0,Y 9.081,Z 695.655,A -85,B 0,C 180,E1 -16059.292,E2 -16059.292} C_VEL
LIN {X 0,Y 21.652,Z 694.059,A -85,B 0,C 180,E1 -16033.152,E2 -16033.152} C_VEL
LIN {X 0,Y 32.785,Z 691.543,A -85,B 0,C 180,E1 -16026.906,E2 -16026.906} C_VEL
LIN {X 0,Y 34.626,Z 691,A -85,B 0,C 180,E1 -16024.957,E2 -16024.957} C_VEL
LIN {X 0,Y 33.643,Z 691.335,A -85,B 0,C 180,E1 -16020.001,E2 -16020.001} C_VEL
LIN {X 0,Y 32.363,Z 691.79,A -85,B 0,C 180,E1 -16015.433,E2 -16015.433} C_VEL
LIN {X 0,Y 21.424,Z 694.292,A -85,B 0,C 180,E1 -16009.775,E2 -16009.775} C_VEL
LIN {X 0,Y 12.503,Z 695.544,A -85,B 0,C 180,E1 -15997.169,E2 -15997.169} C_VEL
LIN {X 0,Y 5.824,Z 696.192,A -85,B 0,C 180,E1 -15930,E2 -15930} C_VEL
LIN {X 0,Y 8.948,Z 695.978,A -85,B 0,C 180,E1 -15878.242,E2 -15878.242} C_VEL
LIN {X 0,Y 19.219,Z 694.714,A -85,B 0,C 180,E1 -15854.312,E2 -15854.312} C_VEL
LIN {X 0,Y 19.219,Z 694.714,A -85,B 0,C 180,E1 -15854.312,E2 -15854.312}

QRS_NEXT_CUT()

QRS_NEXT()
QRS_HOME()

END
